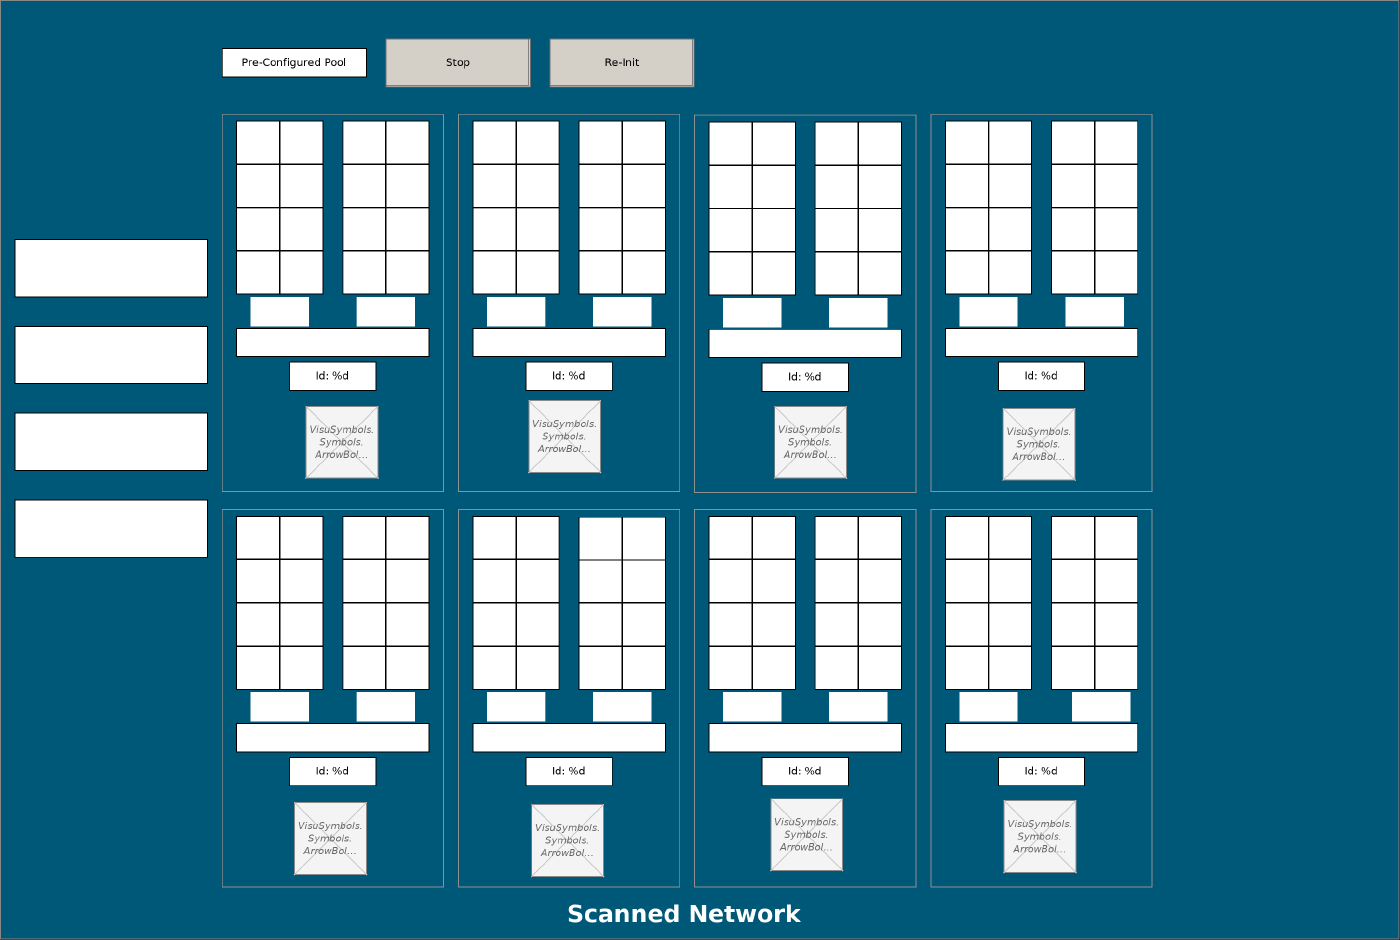
VISUALIZATION Physical  // 1452x975
    RoundedRectangle (0,0 1452x975)
    GroupBox (720,111 230x400), invisible if: GVL_HMI.arrPhysicalMissing[2]
        Rectangle (15,15 45x45), colour toggle: GVL_HMI.arrTerminalData[2][0]
        Rectangle (15,150 45x45), colour toggle: GVL_HMI.arrTerminalData[2][6]
        Rectangle (60,150 45x45), colour toggle: GVL_HMI.arrTerminalData[2][7]
        Rectangle (60,15 45x45), colour toggle: GVL_HMI.arrTerminalData[2][1]
        Rectangle (15,60 45x45), colour toggle: GVL_HMI.arrTerminalData[2][2]
        Rectangle (60,60 45x45), colour toggle: GVL_HMI.arrTerminalData[2][3]
        Rectangle (60,105 45x45), colour toggle: GVL_HMI.arrTerminalData[2][5]
        Rectangle (125,15 45x45), colour toggle: GVL_HMI.arrTerminalData[2][8]
        Rectangle (125,60 45x45), colour toggle: GVL_HMI.arrTerminalData[2][10]
        Rectangle (125,150 45x45), colour toggle: GVL_HMI.arrTerminalData[2][14]
        Rectangle (170,60 45x45), colour toggle: GVL_HMI.arrTerminalData[2][11]
        Rectangle (170,150 45x45), colour toggle: GVL_HMI.arrTerminalData[2][15]
        Rectangle (15,105 45x45), colour toggle: GVL_HMI.arrTerminalData[2][4]
        Rectangle (30,198 60x30), text list: 'RackText', text index: GVL_HMI.arrTerminalNames[4]
        Rectangle (140,198 60x30), text list: 'RackText', text index: GVL_HMI.arrTerminalNames[5]
        Rectangle (170,15 45x45), colour toggle: GVL_HMI.arrTerminalData[2][9]
        Rectangle (125,105 45x45), colour toggle: GVL_HMI.arrTerminalData[2][12]
        Rectangle (170,105 45x45), colour toggle: GVL_HMI.arrTerminalData[2][13]
        Rectangle (70,265 90x30), "Id: %d", text variable: GVL_HMI.arrPhysicalIds[2], colour toggle: GVL_HMI.arrConnected[2]
        Rectangle (15,230 200x30), text list: 'RackText', text index: GVL_HMI.arrRackNames[2]
        Image (83,310 75x75), image: VisuSymbols.Symbols.ArrowBoldRight
    GroupBox (230,520 230x400), invisible if: GVL_HMI.arrPhysicalMissing[4]
        Rectangle (15,15 45x45), colour toggle: GVL_HMI.arrTerminalData[4][0]
        Rectangle (60,15 45x45), colour toggle: GVL_HMI.arrTerminalData[4][1]
        Rectangle (60,105 45x45), colour toggle: GVL_HMI.arrTerminalData[4][5]
        Rectangle (60,150 45x45), colour toggle: GVL_HMI.arrTerminalData[4][7]
        Rectangle (15,60 45x45), colour toggle: GVL_HMI.arrTerminalData[3][2]
        Rectangle (15,105 45x45), colour toggle: GVL_HMI.arrTerminalData[4][4]
        Rectangle (15,150 45x45), colour toggle: GVL_HMI.arrTerminalData[4][6]
        Rectangle (60,60 45x45), colour toggle: GVL_HMI.arrTerminalData[4][3]
        Rectangle (125,15 45x45), colour toggle: GVL_HMI.arrTerminalData[4][8]
        Rectangle (170,15 45x45), colour toggle: GVL_HMI.arrTerminalData[4][9]
        Rectangle (125,60 45x45), colour toggle: GVL_HMI.arrTerminalData[4][10]
        Rectangle (170,60 45x45), colour toggle: GVL_HMI.arrTerminalData[4][11]
        Rectangle (125,105 45x45), colour toggle: GVL_HMI.arrTerminalData[4][12]
        Rectangle (170,105 45x45), colour toggle: GVL_HMI.arrTerminalData[4][13]
        Rectangle (125,150 45x45), colour toggle: GVL_HMI.arrTerminalData[4][14]
        Rectangle (170,150 45x45), colour toggle: GVL_HMI.arrTerminalData[4][15]
        Rectangle (30,198 60x30), text list: 'RackText', text index: GVL_HMI.arrTerminalNames[8]
        Rectangle (140,198 60x30), text list: 'RackText', text index: GVL_HMI.arrTerminalNames[9]
        Rectangle (70,265 90x30), "Id: %d", text variable: GVL_HMI.arrPhysicalIds[4], colour toggle: GVL_HMI.arrConnected[4]
        Rectangle (15,230 200x30), text list: 'RackText', text index: GVL_HMI.arrRackNames[4]
        Image (75,312 75x75), image: VisuSymbols.Symbols.ArrowBoldRight
    GroupBox (475,110 230x400), invisible if: GVL_HMI.arrPhysicalMissing[1]
        Rectangle (15,15 45x45), colour toggle: GVL_HMI.arrTerminalData[1][0]
        Rectangle (60,15 45x45), colour toggle: GVL_HMI.arrTerminalData[1][1]
        Rectangle (60,105 45x45), colour toggle: GVL_HMI.arrTerminalData[1][5]
        Rectangle (60,150 45x45), colour toggle: GVL_HMI.arrTerminalData[1][7]
        Rectangle (15,60 45x45), colour toggle: GVL_HMI.arrTerminalData[1][2]
        Rectangle (15,105 45x45), colour toggle: GVL_HMI.arrTerminalData[1][4]
        Rectangle (15,150 45x45), colour toggle: GVL_HMI.arrTerminalData[1][6]
        Rectangle (60,60 45x45), colour toggle: GVL_HMI.arrTerminalData[1][3]
        Rectangle (125,15 45x45), colour toggle: GVL_HMI.arrTerminalData[1][8]
        Rectangle (170,15 45x45), colour toggle: GVL_HMI.arrTerminalData[1][9]
        Rectangle (125,60 45x45), colour toggle: GVL_HMI.arrTerminalData[1][10]
        Rectangle (170,60 45x45), colour toggle: GVL_HMI.arrTerminalData[1][11]
        Rectangle (125,105 45x45), colour toggle: GVL_HMI.arrTerminalData[1][12]
        Rectangle (170,105 45x45), colour toggle: GVL_HMI.arrTerminalData[1][13]
        Rectangle (125,150 45x45), colour toggle: GVL_HMI.arrTerminalData[1][14]
        Rectangle (170,150 45x45), colour toggle: GVL_HMI.arrTerminalData[1][15]
        Rectangle (30,198 60x30), text list: 'RackText', text index: GVL_HMI.arrTerminalNames[2]
        Rectangle (140,198 60x30), text list: 'RackText', text index: GVL_HMI.arrTerminalNames[3]
        Rectangle (70,265 90x30), "Id: %d", text variable: GVL_HMI.arrPhysicalIds[1], colour toggle: GVL_HMI.arrConnected[1]
        Rectangle (15,230 200x30), text list: 'RackText', text index: GVL_HMI.arrRackNames[1]
        Image (73,305 75x75), image: VisuSymbols.Symbols.ArrowBoldRight
    GroupBox (965,110 230x400), invisible if: GVL_HMI.arrPhysicalMissing[3]
        Rectangle (15,15 45x45), colour toggle: GVL_HMI.arrTerminalData[3][0]
        Rectangle (60,15 45x45), colour toggle: GVL_HMI.arrTerminalData[3][1]
        Rectangle (60,105 45x45), colour toggle: GVL_HMI.arrTerminalData[3][4]
        Rectangle (60,150 45x45), colour toggle: GVL_HMI.arrTerminalData[3][6]
        Rectangle (15,60 45x45), colour toggle: GVL_HMI.arrTerminalData[3][2]
        Rectangle (15,105 45x45), colour toggle: GVL_HMI.arrTerminalData[3][3]
        Rectangle (15,150 45x45), colour toggle: GVL_HMI.arrTerminalData[3][5]
        Rectangle (60,60 45x45), colour toggle: GVL_HMI.arrTerminalData[3][3]
        Rectangle (125,15 45x45), colour toggle: GVL_HMI.arrTerminalData[3][8]
        Rectangle (170,15 45x45), colour toggle: GVL_HMI.arrTerminalData[3][9]
        Rectangle (125,60 45x45), colour toggle: GVL_HMI.arrTerminalData[3][10]
        Rectangle (170,60 45x45), colour toggle: GVL_HMI.arrTerminalData[3][11]
        Rectangle (125,105 45x45), colour toggle: GVL_HMI.arrTerminalData[3][12]
        Rectangle (170,105 45x45), colour toggle: GVL_HMI.arrTerminalData[3][13]
        Rectangle (125,150 45x45), colour toggle: GVL_HMI.arrTerminalData[3][14]
        Rectangle (170,150 45x45), colour toggle: GVL_HMI.arrTerminalData[3][15]
        Rectangle (30,198 60x30), text list: 'RackText', text index: GVL_HMI.arrTerminalNames[6]
        Rectangle (140,198 60x30), text list: 'RackText', text index: GVL_HMI.arrTerminalNames[7]
        Rectangle (70,265 90x30), "Id: %d", text variable: GVL_HMI.arrPhysicalIds[3], colour toggle: GVL_HMI.arrConnected[3]
        Rectangle (15,230 200x30), text list: 'RackText', text index: GVL_HMI.arrRackNames[3]
        Image (75,313 75x75), image: VisuSymbols.Symbols.ArrowBoldRight
    GroupBox (720,520 230x400), invisible if: GVL_HMI.arrPhysicalMissing[6]
        Rectangle (15,15 45x45), colour toggle: MAIN.arrFb1In[0].stRack.ST_In.Input1
        Rectangle (60,15 45x45), colour toggle: MAIN.arrFb1In[0].stRack.ST_In.Input2
        Rectangle (60,105 45x45), colour toggle: MAIN.arrFb1In[0].stRack.ST_In.Input6
        Rectangle (60,150 45x45), colour toggle: MAIN.arrFb1In[0].stRack.ST_In.Input8
        Rectangle (15,60 45x45), colour toggle: MAIN.arrFb1In[0].stRack.ST_In.Input3
        Rectangle (15,105 45x45), colour toggle: MAIN.arrFb1In[0].stRack.ST_In.Input5
        Rectangle (15,150 45x45), colour toggle: MAIN.arrFb1In[0].stRack.ST_In.Input7
        Rectangle (60,60 45x45), colour toggle: MAIN.arrFb1In[0].stRack.ST_In.Input4
        Rectangle (30,198 60x30), text list: 'RackText', text index: GVL_HMI.arrTerminalNames[12]
        Rectangle (70,265 90x30), "Id: %d", text variable: GVL_HMI.arrPhysicalIds[6], colour toggle: GVL_HMI.arrConnected[6]
        Rectangle (125,15 45x45), colour toggle: MAIN.arrFb1In[0].stRack.ST_In.Input1
        Rectangle (140,198 60x30), text list: 'RackText', text index: GVL_HMI.arrTerminalNames[13]
        Rectangle (170,15 45x45), colour toggle: MAIN.arrFb1In[0].stRack.ST_In.Input2
        Rectangle (170,105 45x45), colour toggle: MAIN.arrFb1In[0].stRack.ST_In.Input6
        Rectangle (170,150 45x45), colour toggle: MAIN.arrFb1In[0].stRack.ST_In.Input8
        Rectangle (125,60 45x45), colour toggle: MAIN.arrFb1In[0].stRack.ST_In.Input3
        Rectangle (125,105 45x45), colour toggle: MAIN.arrFb1In[0].stRack.ST_In.Input5
        Rectangle (125,150 45x45), colour toggle: MAIN.arrFb1In[0].stRack.ST_In.Input7
        Rectangle (170,60 45x45), colour toggle: MAIN.arrFb1In[0].stRack.ST_In.Input4
        Rectangle (15,230 200x30), text list: 'RackText', text index: GVL_HMI.arrRackNames[6]
        Image (79,308 75x75), image: VisuSymbols.Symbols.ArrowBoldRight
    GroupBox (230,110 230x400), invisible if: GVL_HMI.arrPhysicalMissing[0]
        Rectangle (15,15 45x45), colour toggle: GVL_HMI.arrTerminalData[0][0]
        Rectangle (60,15 45x45), colour toggle: GVL_HMI.arrTerminalData[0][1]
        Rectangle (60,105 45x45), colour toggle: GVL_HMI.arrTerminalData[0][5]
        Rectangle (60,150 45x45), colour toggle: GVL_HMI.arrTerminalData[0][7]
        Rectangle (15,60 45x45), colour toggle: GVL_HMI.arrTerminalData[0][2]
        Rectangle (15,105 45x45), colour toggle: GVL_HMI.arrTerminalData[0][4]
        Rectangle (15,150 45x45), colour toggle: GVL_HMI.arrTerminalData[0][6]
        Rectangle (60,60 45x45), colour toggle: GVL_HMI.arrTerminalData[0][3]
        Rectangle (125,15 45x45), colour toggle: GVL_HMI.arrTerminalData[0][8]
        Rectangle (125,60 45x45), colour toggle: GVL_HMI.arrTerminalData[0][10]
        Rectangle (170,60 45x45), colour toggle: GVL_HMI.arrTerminalData[0][11]
        Rectangle (125,105 45x45), colour toggle: GVL_HMI.arrTerminalData[0][12]
        Rectangle (170,105 45x45), colour toggle: GVL_HMI.arrTerminalData[0][13]
        Rectangle (125,150 45x45), colour toggle: GVL_HMI.arrTerminalData[0][14]
        Rectangle (170,150 45x45), colour toggle: GVL_HMI.arrTerminalData[0][15]
        Rectangle (30,198 60x30), text list: 'RackText', text index: GVL_HMI.arrTerminalNames[0]
        Rectangle (140,198 60x30), text list: 'RackText', text index: GVL_HMI.arrTerminalNames[1]
        Rectangle (70,265 90x30), "Id: %d", text variable: GVL_HMI.arrPhysicalIds[0], colour toggle: GVL_HMI.arrConnected[0]
        Rectangle (15,230 200x30), text list: 'RackText', text index: GVL_HMI.arrRackNames[0]
        Rectangle (170,15 45x45), colour toggle: GVL_HMI.arrTerminalData[0][9]
        Image (87,311 75x75), image: VisuSymbols.Symbols.ArrowBoldRight
    GroupBox (475,520 230x400), invisible if: GVL_HMI.arrPhysicalMissing[5]
        Rectangle (15,15 45x45), colour toggle: GVL_HMI.arrTerminalData[5][0]
        Rectangle (60,15 45x45), colour toggle: GVL_HMI.arrTerminalData[5][1]
        Rectangle (60,105 45x45), colour toggle: GVL_HMI.arrTerminalData[5][5]
        Rectangle (60,150 45x45), colour toggle: GVL_HMI.arrTerminalData[5][7]
        Rectangle (15,60 45x45), colour toggle: GVL_HMI.arrTerminalData[5][2]
        Rectangle (15,105 45x45), colour toggle: GVL_HMI.arrTerminalData[5][4]
        Rectangle (15,150 45x45), colour toggle: GVL_HMI.arrTerminalData[5][6]
        Rectangle (60,60 45x45), colour toggle: GVL_HMI.arrTerminalData[5][3]
        Rectangle (125,60 45x45), colour toggle: GVL_HMI.arrTerminalData[5][10]
        Rectangle (170,60 45x45), colour toggle: GVL_HMI.arrTerminalData[5][11]
        Rectangle (125,105 45x45), colour toggle: GVL_HMI.arrTerminalData[5][12]
        Rectangle (170,105 45x45), colour toggle: GVL_HMI.arrTerminalData[5][13]
        Rectangle (125,150 45x45), colour toggle: GVL_HMI.arrTerminalData[5][14]
        Rectangle (170,150 45x45), colour toggle: GVL_HMI.arrTerminalData[5][15]
        Rectangle (30,198 60x30), text list: 'RackText', text index: GVL_HMI.arrTerminalNames[10]
        Rectangle (140,198 60x30), text list: 'RackText', text index: GVL_HMI.arrTerminalNames[11]
        Rectangle (170,16 45x45), colour toggle: GVL_HMI.arrTerminalData[5][9]
        Rectangle (125,16 45x45), colour toggle: GVL_HMI.arrTerminalData[5][8]
        Rectangle (70,265 90x30), "Id: %d", text variable: GVL_HMI.arrPhysicalIds[5], colour toggle: GVL_HMI.arrConnected[5]
        Rectangle (15,230 200x30), text list: 'RackText', text index: GVL_HMI.arrRackNames[5]
        Image (76,314 75x75), image: VisuSymbols.Symbols.ArrowBoldRight
    GroupBox (965,520 230x400), invisible if: GVL_HMI.arrPhysicalMissing[7]
        Rectangle (15,15 45x45), colour toggle: MAIN.arrFb1In[1].stRack.ST_In.Input1
        Rectangle (60,15 45x45), colour toggle: MAIN.arrFb1In[1].stRack.ST_In.Input2
        Rectangle (60,105 45x45), colour toggle: MAIN.arrFb1In[1].stRack.ST_In.Input6
        Rectangle (60,150 45x45), colour toggle: MAIN.arrFb1In[1].stRack.ST_In.Input8
        Rectangle (15,60 45x45), colour toggle: MAIN.arrFb1In[1].stRack.ST_In.Input3
        Rectangle (15,105 45x45), colour toggle: MAIN.arrFb1In[1].stRack.ST_In.Input5
        Rectangle (15,150 45x45), colour toggle: MAIN.arrFb1In[1].stRack.ST_In.Input7
        Rectangle (60,60 45x45), colour toggle: MAIN.arrFb1In[1].stRack.ST_In.Input4
        Rectangle (30,198 60x30), text list: 'RackText', text index: GVL_HMI.arrTerminalNames[14]
        Rectangle (70,265 90x30), "Id: %d", text variable: GVL_HMI.arrPhysicalIds[7], colour toggle: GVL_HMI.arrConnected[7]
        Rectangle (125,15 45x45), colour toggle: MAIN.arrFb1In[1].stRack.ST_In.Input1
        Rectangle (147,198 60x30), text list: 'RackText', text index: GVL_HMI.arrTerminalNames[15]
        Rectangle (15,230 200x30), text list: 'RackText', text index: GVL_HMI.arrRackNames[7]
        Rectangle (170,15 45x45), colour toggle: MAIN.arrFb1In[1].stRack.ST_In.Input2
        Rectangle (170,105 45x45), colour toggle: MAIN.arrFb1In[1].stRack.ST_In.Input6
        Rectangle (170,150 45x45), colour toggle: MAIN.arrFb1In[1].stRack.ST_In.Input8
        Rectangle (125,60 45x45), colour toggle: MAIN.arrFb1In[1].stRack.ST_In.Input3
        Rectangle (125,105 45x45), colour toggle: MAIN.arrFb1In[1].stRack.ST_In.Input5
        Rectangle (125,150 45x45), colour toggle: MAIN.arrFb1In[1].stRack.ST_In.Input7
        Rectangle (170,60 45x45), colour toggle: MAIN.arrFb1In[1].stRack.ST_In.Input4
        Image (76,310 75x75), image: VisuSymbols.Symbols.ArrowBoldRight
    Rectangle (230,50 150x30), "Pre-Configured Pool"
        OnMouseDown: change screen: Configured
    Rectangle (15,248 200x60), colour toggle: GVL_HMI.bType1Present, text list: 'RackText', text index: 11
    Rectangle (15,338 200x60), colour toggle: GVL_HMI.bType2Present, text list: 'RackText', text index: 8
    Rectangle (15,428 200x60), colour toggle: GVL_HMI.bType3Present, text list: 'RackText', text index: 9
    Rectangle (15,518 200x60), colour toggle: GVL_HMI.bType4Present, text list: 'RackText', text index: 10
    Button (400,40 150x50), "Stop"
        toggle MAIN.bStop
    Button (570,40 150x50), "Re-Init"
        tap MAIN.bReset
    Label (228,933 963x30), "Scanned Network"
END_VISUALIZATION

(* stored: Version 1.1.0.1, ProductVersion 3.1.4024.6
   Visu Physical: Id {5e5ec2d5-fafd-47ed-836a-7586d2bfe36a} *)
